TYPE ST_HW_InputsTurnTableDTU :

STRUCT
	TT						: ST_HW_InputsTT; //Turning inputs	
	CV						: ST_HW_InputsTTConv; //Drive/Transport control sensors
	Sensor_Overhang_12		: BOOL; // Sensor overhang axis 1-2 forward	
	Sensor_Overhang_21		: BOOL; // Sensor overhang axis 2-1 reverse
	Sensor_Overhang_34		: BOOL; // Sensor overhang axis 3-4 forward
	Sensor_Overhang_43		: BOOL; // Sensor overhang axis 4-3 reverse
	Sensor_Pos_Down			: BOOL; // Sensor position lift down
	Sensor_Pos_Up			: BOOL; // Sensor position lift up				
END_STRUCT
END_TYPE

(* stored: Version 1.1.0.1, ProductVersion 3.1.4022.12
   DUT ST_HW_InputsTurnTableDTU: Id {c444ceda-6bb5-41d8-87d0-a9a9ba846663} *)
